{attribute 'qualified_only'}
VAR_GLOBAL
	stControlParams : ST_BoxParams; 
END_VAR

(* stored: Version 1.1.0.1, ProductVersion 3.1.4024.12
   GVL GVL_ControlBox: Id {befa822b-95e2-4d5b-8b35-a19e7f4b9a6c} *)
